Staubli VAL3: modIMM.pjx

--- modIMM.pjx ---
Parameters version=s7.2 stackSize=5000 millimeterUnit=true
Program file=_StartMachine.pgx
Program file=_WaitAuto.pgx
Program file=_WaitEnd.pgx
Program file=_WaitPart.pgx
Program file=_WaitPartDyn.pgx
Program file=BtRobotOff.pgx
Program file=checkMotStack.pgx
Program file=childAction.pgx
Program file=getSetting.pgx
Program file=IMMTiming.pgx
Program file=init.pgx
Program file=loadLibraries.pgx
Program file=primeAreaTest.pgx
Program file=primeMotStack.pgx
Program file=registerSetting.pgx
Program file=retrieveViews.pgx
Program file=runHigh.pgx
Program file=runLow.pgx
Program file=secuTask1.pgx
Program file=secuTask2.pgx
Program file=setDryRunSig.pgx
Program file=setSetting.pgx
Program file=slot.pgx
Program file=start.pgx
Program file=startAreaTest.pgx
Program file=stop.pgx
Program file=stopAreaTest.pgx
Program file=taskPartMade.pgx
Program file=updateView.pgx
Program file=WaitPart.pgx
Data file=modIMM.dtx
Library alias=io path=Disk://io/io.pjx
Library alias=SYS path=Disk://io_System/io_System.pjx
Library alias=scr path=Disk://Plastic/coreModules/modScreen/modScreen.pjx
Library alias=str path=Disk://Libraries/stringHandling/stringHandling.pjx
Library alias=lang path=Disk://Plastic/i18n/i18n.pjx
Library alias=debug path=Disk://Libraries/debug/debug.pjx
Library alias=data path=Disk://zData/zData.pjx
Library alias=status path=Disk://Plastic/coreModules/modStatusModel/modStatusModel.pjx
Library alias=EV path=Disk://Plastic/Consts/EVENT/EVENT.pjx
Library alias=sig path=Disk://Plastic/coreModules/modSignalSlot/modSignalSlot.pjx
Library alias=STATE path=Disk://Plastic/Consts/STATE/STATE.pjx
Library alias=views path=Disk://Plastic/coreModules/viewContainer/viewContainer.pjx
Library alias=jt path=Disk://Libraries/jointFunctions/jointFunctions.pjx
Type name=event path=Disk://Plastic/Types/event/event.pjx
Type name=settingType path=Disk://Plastic/Types/setting/setting.pjx
Type name=viewType path=Disk://Plastic/Types/view/view.pjx
Type name=childNodeType path=Disk://Plastic/Types/childNode/childNode.pjx
Type name=nodeType path=Disk://Plastic/Types/node/node.pjx

--- start.pgx ---
public program start()
begin
  // set nCaseBtRobOff to 1 instead of 0 in order to initialize the robot off function properly
  // If nCaseBtRobOff is 0 at start up it may happen that SYS:doRobotOff["+toString("",moduleIndex)+"] is on although btRobotOff assumes that
  // SYS:doRobotOff["+toString("",moduleIndex)+"] is off.

  call debug:setVerbosity(libPath(),debug:LEV_INFO)
  call loadLibraries()
  // call setDryRunSig(data:setDryRun)
  call sig:connect(EV:DRY_RUN,libPath())
  call sig:connect(EV:FATAL_ERROR,libPath())
  call sig:connect(EV:START_COMPLETE,libPath())
  call status:registerStatus(libPath(),status:CL_STATUS,"Wait for mould free condition","SYS:doMouldFree["+toString("",moduleIndex)+"]==true","SYS:doMouldFree["+toString("",moduleIndex)+"]==false",false,WAIT_MOULD_FREE,false)
  call status:registerStatus(libPath(),status:CL_STATUS,"Wait for mould open","SYS:diMouldOpen["+toString("",moduleIndex)+"]==true","SYS:diMouldOpen["+toString("",moduleIndex)+"]==false",false,WAIT_MOULD_OPEN,false)
  call status:registerStatus(libPath(),status:CL_STATUS,"Wait for robot enabled","SYS:doRobotOff["+toString("",moduleIndex)+"]==false","SYS:doRobotOff["+toString("",moduleIndex)+"]==true",false,WAIT_ROB_ENABLE,false)
  call status:registerStatus(libPath(),status:CL_STATUS,"Wait for IMM in auto mode","SYS:diMachineInAuto["+toString("",moduleIndex)+"]==true","SYS:diMachineInAuto["+toString("",moduleIndex)+"]==false",false,WAIT_ROB_ENABLE,false)
  call status:registerStatus(libPath(),status:CL_STATUS,"Wait for part produced","SYS:bPartMade["+toString("",moduleIndex)+"]==true","SYS:bPartMade["+toString("",moduleIndex)+"]==false",false,WAIT_PARTMADE,false)
  call status:registerStatus(libPath(),status:CL_ERROR,"Mould area test failed. Robot was not programmed to enter mould","","",true,AREA_TEST_FAIL,true)
  call status:registerStatus(libPath(),status:CL_ERROR,"Home position is defined in mould area","","",true,HOME_IN_MOULD,true)
  call status:registerStatus(libPath(),status:CL_ERROR,"Arm in mould while mould is not open","","",true,ARM_IN_MOULD_NO,true)
  call status:registerStatus(libPath(),status:CL_ERROR,"Arm in mould while 'Enable Closure' signal is set","","",true,ARM_IN_MOULD_ST,true)
end

--- _StartMachine.pgx ---
public program _StartMachine()
// Start machine cycle
  local bool bAreaTest
  local num nOldSpeedScale
  local bool bTestRun
  local string txt
  local num time
  local string sValue
begin
  //
  // add list of pending status messages
  //!i18n 16 -> "Wait for Mould Free Condition"

  call status:setEnabled(WAIT_MOULD_FREE,true)
  //!change 23.05.06, vdg: reduce speed in test mode when approaching the mould area boundary
  // from inside towards outside
  //!change 08.09.06, vdg: store data:setTestRun in a local variable
  bTestRun=data:setTestRun
  // prime the motion stack monitor which checks if the arm is actually
  // programmed to leave the mould when StartMachine() is called
  call primeMotStack()
  if bTestRun
    //wait(secu:nSafeZoneDist[0]<300)
    nOldSpeedScale=getMonitorSpeed()
    //!fix 09.06.06, vdg: set speed to the lower speed setting (current speedScale() or dry run speed)
    ///TODO
    //$setSpeed(min(speedScale(),10))
    //call setSpeed(min(getMonitorSpeed(),10))
    //wait(secu:nSafeZoneDist[0]<50)
    //$setSpeed(1)
    ///TODO
    //call setSpeed(1)
  endIf
  // WAIT GRIPPER OUT OF MOULD AREA ==================================================================================
  // record the safety distance of the robot

  time=clock()
  //requiredTime=0.2
  //currentTime=0
  // if (speedScale()>99) and (workingMode()==4) and (SYS:diMachineInAuto[moduleIndex]==true) and !bTestRun
  if (getMonitorSpeed()>99) and (workingMode()==4) and !bTestRun
    do
      // Check if there are still motions in the stack.
      // If it is empty, it means the robot never leaves the mould area before
      // StartMachine() is called.
      call checkMotStack()
    until (SYS:doMouldFree[moduleIndex]==true)
  else
    do
      // Check if there are still motions in the stack.
      // If it is empty, it means the robot never leaves the mould area before
      // StartMachine() is called.
      call checkMotStack()
    until (SYS:doMouldFree[moduleIndex]==true)
  endIf
  //
  call status:setEnabled(WAIT_MOULD_FREE,false)
  //
  //!change 18.05.06, vdg: check if doMouldFree has toggled
  call stopAreaTest(bAreaTest)
  // START MACHINE CYCLE =============================================================================================
  //!change 16.02.06, vdg: Allow to start IMM in endIf cycle mode SYS:bStartInEndCycl is set
  if (!SYS:CE_Requested or SYS:bStartInEndCycl) and !SYS:bPartMade[moduleIndex] and bAreaTest
    //!change 18.05.06, vdg: Stop robot at point where machine is being started
    //  and ask the user if it is safe to start the IMM
    if bTestRun
      bSuspendForTest=true
      // reset original speedScale only if speed was not modified by user meanwhile
      // wait for settled arm
      watch(isSettled(),3)
      // reset old speed setting if it wasn't changed by the user
      if getMonitorSpeed()==1
        ///TODO
        //$setSpeed(nOldSpeedScale)
        //call setSpeed(nOldSpeedScale)
      endIf
      //sValue=toString("4.0",secu:nSafeZoneDist[0])
      call str:printf((("Robot stopped approx. at point where IMM cycle is being started (Overshoot: %1mm). Press START to continue!")),sValue,txt)
      ///TODO
      //call ui:popUpCond(txt,"SYS:bBtStart==true",false)
      bSuspendForTest=true
      wait(bSuspendForTest==false)
    endIf
    //!change 08.06.06, vdg: Start IMM only if dry run mode is not active
    if !bTestRun
      SYS:doStartMachine[moduleIndex]=true
    endIf
    //call stat:stopTakeTime()
    //call stat:stopCycleTime()
    //call stat:startCycleTime()
    //call stat:startRobotTime()
  endIf
  //
end

--- _WaitAuto.pgx ---
public program _WaitAuto()
// Wait here until the machine is prepared to be started
begin
  // Enable Robot Off function........................................................
  bRobotOffAllow=true
  //
  //!change 18.06.05, vdg: Prime area test
  call primeAreaTest()
  //
  // ignore messages if in dry run mode
  if data:setDryRun==false
    call status:setEnabled(WAIT_IMM_AUTO,true)
  endIf
  call status:setEnabled(WAIT_MOULD_OPEN,true)
  call status:setEnabled(WAIT_ROB_ENABLE,true)
  // Stop the robot cycle time timer
  //call stat:stopRobotTime()
  // Wait machine in AUTO.............................................................
  do
    //Robot in position to be able use the Robot Off function.
    if SYS:diMachineInAuto[moduleIndex]==false and SYS:bRobotOffCalled[moduleIndex]
      bAtWaitPosition=true
    endIf
    //!change 08.06.06, vdg: ignore automatic signal in dry run mode
  until ((SYS:diMachineInAuto[moduleIndex]==true or data:setDryRun==true) and SYS:diMouldOpen[moduleIndex]==true and bRobotOff==false)
  //
  // Robot not in position to use Robot Off function..................................
  bAtWaitPosition=false
  //
  call status:setEnabled(WAIT_IMM_AUTO,false)
  call status:setEnabled(WAIT_MOULD_OPEN,false)
  call status:setEnabled(WAIT_ROB_ENABLE,false)
  //
  // Start measuring the take out time
  //call stat:startTakeTime()
  //
  call startAreaTest()
end

--- _WaitEnd.pgx ---
public program _WaitEnd()
// Halt robot here if "END" is activated
  local num nStateWaitEnd
begin
  // WAIT END OF CYCLE......................................................
  if SYS:CE_Requested and !SYS:bPartMade[moduleIndex] and SYS:doStartMachine[moduleIndex]==false
    do
      // Robot is running in production cycle (StateRobot==10)
      if SYS:nStateRobot==10 and isPowered() and SYS:diMachineInAuto[moduleIndex]==true
        // "End Of Cycle" running and no more parts in mould
        if SYS:CE_Requested and !SYS:bPartMade[moduleIndex] and SYS:diMachineInAuto[moduleIndex]==true
          nStateWaitEnd=30
        endIf
        // Robot Off called
        if SYS:bRobotOffCalled[moduleIndex]
          nStateWaitEnd=40
        endIf
      else
        // Robot or Machine not in AUTO
        if SYS:nStateRobot!=10
          nStateWaitEnd=0
        else
          // "End Of Cycle" running and no more parts in mould
          if SYS:CE_Requested and !SYS:bPartMade[moduleIndex] and SYS:CE_AtEndPos==false
            nStateWaitEnd=30
          endIf
          // Robot Off called
          if SYS:bRobotOffCalled[moduleIndex] and !bAtWaitPosition
            nStateWaitEnd=40
          endIf
        endIf
      endIf
      //
      switch (nStateWaitEnd)
        //
        //  Robot and Machine not in Auto.......................................
        case 0
          if SYS:diMachineInAuto[moduleIndex]==false
            //Wait Machine In Auto
            //user:sMessage[0]=user:sMessage[0]
          else
            //Wait [START] Robot
            //user:sMessage[0]=user:sMessage[0]
          endIf
        break
        //
        // "End Of Cycle" called and no more parts in mould.....................
        case 30
          if SYS:CE_Requested==true and SYS:bPartMade[moduleIndex]==false
            stopMove()
            wait(isSettled())
            SYS:CE_AtEndPos=true
            delay(0)
          endIf
        break
        //
        // Robot Off called.......................................................
        case 40
          wait(isSettled())
          stopMove()
          bAtWaitPosition=true
          delay(0)
        break
      endSwitch
      //
      // Wait until robot is at end position......................................
    until (SYS:CE_AtEndPos==true or bAtWaitPosition==true and isSettled())
    //
    // Reset StartMachine.................................................................................................
    SYS:doStartMachine[moduleIndex]=false
  endIf
end

--- _WaitPartDyn.pgx ---
public program _WaitPartDyn()
// Wait part made in machine and mould fully open
begin
  //!brief
  // Wait for a part being made and conditions for the robot to enter mold.
  //
  call WaitPart(true)
end

--- init.pgx ---
public program init()
  local bool ok
  local string path
  local num idx
begin
  // set module index
  path=libPath()
  path=right(path,1)
  path=toNum(path,moduleIndex,ok)
  if !ok
    moduleIndex=0
  endIf
  name="IMM"+toString("1.0",moduleIndex)
  IMM_IO_PTH="2:IO/1:"+name
  nCaseBtRobOff=1
  bState=false
  pointer=0
  for idx=0 to size(timings)-1
    timings[idx]=0
  endFor

end

--- loadLibraries.pgx ---
program loadLibraries()
begin
//  nResult=scr:libLoad("Plastic/Modules/modScreen.zip","a81d706f651db0a6b2")
//  if nResult!=0
//    name=libPath()
//    nResult=scr:libLoad("Plastic/Modules/modScreen")
//    if nResult!=0
//      popUpMsg(name+":  Problem loading library for scr:")
//      call debug:error(libPath(),": Problem loading library for scr:")
//    else
//      call debug:info(libPath(),": Loading uncrypted version "+scr:libPath())
//    endIf
//  endIf
  // SECU
//  nResult=secu:libLoad("Plastic/Modules/modSafety.zip","a81d706f651db0a6b2")
//  if nResult!=0
//    name=libPath()
//    nResult=secu:libLoad("Plastic/Modules/modSafety")
//    if nResult!=0
//      popUpMsg(name+":  Problem loading library for secu:")
//      call debug:error(libPath(),": Problem loading library for secu:")
//    else
//      call debug:info(libPath(),": Loading uncrypted version "+secu:libPath())
//    endIf
//  endIf
//  // STATUS
//  nResult=stat:libLoad("Plastic/Modules/modStatus.zip","a81d706f651db0a6b2")
//  if nResult!=0
//    name=libPath()
//    nResult=stat:libLoad("Plastic/Modules/modStatus")
//    if nResult!=0
//      popUpMsg(name+":  Problem loading library for stat:")
//      call debug:error(libPath(),": Problem loading library for stat:")
//    else
//      call debug:info(libPath(),": Loading uncrypted version "+stat:libPath())
//    endIf
//  endIf
end

--- primeAreaTest.pgx ---
public program primeAreaTest()
begin
  // reset test state machine
  nAreaTestState=0
end

--- retrieveViews.pgx ---
public program retrieveViews(viewType& view_, num& idx_)
begin
  switch idx_
    case 0
      view_.path=IMM_IO_PTH
      view_.label="IMM"
      call views:appendNode(view_.nodes,"Safety")
      call views:appendNode(view_.nodes,"Machine")
      call views:appendNode(view_.nodes,"Ejectors")
      call views:appendNode(view_.nodes,"Cores")
      call views:appendNode(view_.nodes,"Mould")
      view_.type=view_.TYPE_TREEVIEW
    break
  endSwitch
end

--- run.pgx ---
public program run()
begin
  call taskPartMade()
  call IMMTiming()
end

--- runHigh.pgx ---
public program runHigh()
begin
  call taskPartMade()
  call IMMTiming()
   call BtRobotOff()

  call secuTask1()
  call secuTask2()
end

--- secuTask1.pgx ---
public program secuTask1()
// Control "Mould Area Free" from robot
  local point pLocFlange
  local point pLocTCP
begin
  //
  //!change 23.04.06, vdg: added global variable that contains the distance to the safety zone
  // Security zon in millimeter for wrist relativ to IMM Backside...........
  // nSafeZon[0]=300
  //
  // LOOP: task "RobSafe1"..................................................

    //
    // Get current robot position relative to the frame of IMM Backside.....
    pLocFlange=here(flange,data:fAreaIMM)
    pLocTCP=here(data:tTCP,data:fAreaIMM)
    //
    // Set signal "Mould Area Free" to machine..............................
    nMouldAreaDist=max(pLocTCP.trsf.z,pLocFlange.trsf.z)-nMouldAreaZone
    SYS:doMouldFree[moduleIndex]=nMouldAreaDist<0
    //
    if SYS:doMouldFree==false
      SYS:doStartMachine=false
      bRobotOff=false
    endIf
    //
    //!change 18.05.06, vdg: Test if MouldFree Signal has toggled while robot was in mould
    switch nAreaTestState
      // initialize test
      case 0
        //nAreaTestState=0
        //bAreaFlag=SYS:doMouldFree
      break
      // wait for high state
      case 10
        if SYS:doMouldFree==true
          nAreaTestState=20
        endIf
      break
      // wait for low state
      case 20
        if SYS:doMouldFree==false
          nAreaTestState=30
        endIf
      break
      // wait for high state again
      case 30
        if SYS:doMouldFree==true
          nAreaTestState=40
        endIf
      break
      // final state
      // this state must be reached when startIMM() is called
      case 40
      break
    endSwitch
//  SYS:doSecu[0]=false
//  SYS:doSecu[1]=false
end

--- secuTask2.pgx ---
public program secuTask2()
// Control of Safety realay
  local point pLocFlange
  local point pLocTCP
begin
  // wait until system is initialized
  if SYS:nStateRobot<=STATE:INITIALIZING
    return
  endIf
  if SYS:doSecu[0]==false or SYS:doSecu[1]==false
    return
  endIf
  // Get home position relative to the frame of IMM mould area.....
  if jt:isTXRobot
    pLocFlange=jointToPoint(flange,data:fAreaIMM,data:jHomeTX)
    pLocTCP=jointToPoint(data:tTCP,data:fAreaIMM,data:jHomeTX)
  else
    pLocFlange=jointToPoint(flange,data:fAreaIMM,data:jHomeTS)
    pLocTCP=jointToPoint(data:tTCP,data:fAreaIMM,data:jHomeTS)
  endIf
//
  if pLocTCP.trsf.z>nMouldAreaZone
    call status:raise(HOME_IN_MOULD,"")
  endIf
  // Get current robot position relative to the frame of IMM Backside.....
  pLocFlange=here(flange,data:fAreaIMM)
  pLocTCP=here(data:tTCP,data:fAreaIMM)
  nMouldAreaDist=max(pLocTCP.trsf.z,pLocFlange.trsf.z)-nMouldAreaZone
  //
  // Robotarm in mould when sig:MouldOpen missing or sig:StartIMM is active..........................................................
  if SYS:doMouldFree==false and (SYS:diMouldMidOpen==false and SYS:diMouldOpen==false)
    call status:raise(ARM_IN_MOULD_NO,"")
  endIf
  if (SYS:doMouldFree==false and SYS:doStartMachine==true)
    call status:raise(ARM_IN_MOULD_ST,"")
  endIf
end

--- setDryRunSig.pgx ---
public program setDryRunSig(bool enable_)
begin
  if enable_
    call debug:warning(libPath(),"Dry run mode enabled")
    dioLink(SYS:diEjcIn,SYS:doEjcIn)
    dioLink(SYS:diEjcOut,SYS:doEjcOut)
    dioLink(SYS:diCore1Pos1,SYS:doCore1Pos1)
    dioLink(SYS:diCore1Pos2,SYS:doCore1Pos2)
    dioLink(SYS:diCore2Pos1,SYS:doCore2Pos1)
    dioLink(SYS:diCore2Pos2,SYS:doCore2Pos2)
  else
    call debug:warning(libPath(),"Dry run mode disabled")
    call SYS:InitSysIO()
  endIf
end

--- slot.pgx ---
public program slot(event& event_)
begin
  switch event_.nType
    case EV:DRY_RUN
      call setDryRunSig(event_.sParam=="1")
    break
    case EV:START_COMPLETE
      SYS:doSecu[0]=true
    SYS:doSecu[1]=true
    break
  endSwitch
end

--- stopAreaTest.pgx ---
public program stopAreaTest(bool& bResult_[])
begin
  // test result of area test state machine
  // the state nAreaTestState must be 40
  if nAreaTestState!=40 and nAreaTestState!=0
    call status:raise(AREA_TEST_FAIL,"")
  endIf
  bResult_=nAreaTestState==40 or nAreaTestState==0
end

--- taskPartMade.pgx ---
program taskPartMade()
// Part produced in an IMM
begin
  // Conditions for part made is registered in program.
  // Arm will enter mould. Close mould is not allowed.
  if !bRobotOffAllow
    SYS:doStartMachine[moduleIndex]=false
  endIf
  if SYS:doMouldFree[moduleIndex]==false or SYS:bRobotHome
    bRobotOffAllow=true
  endIf
  // RESET StartMachine.......................................................
  // handle reset according to given IMM type
  switch nImmType
    // standard IMM, e.g. Netstal
    case 0
      // reset doStartMachine when IMM is switched to manual
      if SYS:diMachineInAuto[moduleIndex]==false
        SYS:doStartMachine[moduleIndex]=false
      endIf
      // set robot off signal to IMM
      SYS:doRobotOff[moduleIndex]=bRobotOff
    break
    // IMMs of type 1, that need special treatment of doStartIMM, e.g. Negri Bossi
    case 1
      // reset doStartMachine when IMM is switched to manual and handling is disabled
      if SYS:diMachineInAuto[moduleIndex]==false and SYS:doRobotOff[moduleIndex]==false
        SYS:doStartMachine[moduleIndex]=false
      endIf
      if bRobotOff==true
        // Disable doStartMachine and doRobotOff if the robot is approaching the mold
        // The distance 20mm is set in order to have a pre warning before the arm
        // actually enters the mold area.
        if nMouldAreaDist>-20
          SYS:doStartMachine[moduleIndex]=false
          SYS:doRobotOff[moduleIndex]=false
        else
          SYS:doStartMachine[moduleIndex]=true
          // set robot off signal to IMM
          SYS:doRobotOff[moduleIndex]=bRobotOff
        endIf
      else
        // set robot off signal to IMM
        SYS:doRobotOff[moduleIndex]=bRobotOff
      endIf
    break
  endSwitch

  // RESET PartMade (Ejecor and "Robot OFF")..................................
  if SYS:diMachineInAuto[moduleIndex]==false or bRobotOff==true
    if SYS:diMachineInAuto[moduleIndex]==false
      SYS:doEjcIn=true
      SYS:doEjcOut=true
    else
      SYS:doEjcIn=false
      SYS:doEjcOut=false
    endIf
    switch nStateRstPart[0]
      case 0
        if (SYS:diEjcOut==true and SYS:diEjcIn==false)
          nStateRstPart[0]=1
        endIf
      break
      case 1
        if (SYS:diEjcOut==false and SYS:diEjcIn==true)
          SYS:bPartMade[moduleIndex]=false
          nStateRstPart[0]=0
        endIf
      break
    endSwitch
  else
    nStateRstPart[0]=0
  endIf
  //
  // RESET PartMade (Core and "Robot OFF")...................................
  if SYS:diMachineInAuto[moduleIndex]==false or bRobotOff==true
    if SYS:diMachineInAuto[moduleIndex]==false
      SYS:doCore1Pos1=true
      SYS:doCore1Pos2=true
    else
      SYS:doCore1Pos1=false
      SYS:doCore1Pos2=false
    endIf
    switch nStateRstPart[1]
      case 0
        if (SYS:diCore1Pos2==true and SYS:diCore1Pos1==false)
          nStateRstPart[1]=1
        endIf
      break
      case 1
        if (SYS:diCore1Pos2==false and SYS:diCore1Pos1==true)
          SYS:bPartMade[moduleIndex]=false
          nStateRstPart[1]=0
        endIf
      break
    endSwitch
  else
    nStateRstPart[1]=0
  endIf
  //
  // RESET PartMade (machine goes from manual mode to auto)..................
  switch nStateRstPart[3]
    case 0
      if (SYS:diMachineInAuto[moduleIndex]==false)
        nStateRstPart[3]=1
      endIf
    break
    case 1
      if (SYS:diMachineInAuto[moduleIndex]==true)
        SYS:bPartMade[moduleIndex]=false
        SYS:doEjcIn=false
        SYS:doEjcOut=false
        SYS:doCore1Pos1=false
        SYS:doCore1Pos2=false
        nStateRstPart[3]=0
      endIf
    break
  endSwitch
  //
  // PART MADE.............................................................
  switch nStatePartMade
    // Mould open
    case 0
      if (SYS:bPartMade[moduleIndex]==false and SYS:diMouldOpen[moduleIndex]==true and SYS:diMachineInAuto[moduleIndex]==true)
        nStatePartMade=1
        // count parts
        data:cyclesProduced=data:cyclesProduced+1
        if SYS:diRejectPart==true
          data:cyclesRejected=data:cyclesRejected+1
        endIf
      endIf
    break
    // Mould is closing
    case 1
      if SYS:diMouldOpen[moduleIndex]==false and SYS:diMachineInAuto[moduleIndex]==true
        nStatePartMade=2
      endIf
    break
    // Mould closed
    case 2
      if SYS:diMouldClosed[moduleIndex]==true and SYS:diMachineInAuto[moduleIndex]==true
        SYS:bPartMade[moduleIndex]=true
        // Reset of ejector signals disabled here, as some IMMs
        // have problems when ejector signal is reset when mould is closed as the ejectors
        // are not held in position actively anymore (due to leacking valve or similar).
        // Instead the ejector signals are reset when the mould starts opening again
        // (see state 3)
        //SYS:doEjcIn=false
        //SYS:doEjcOut=false
        SYS:doStartMachine[moduleIndex]=false
        nStatePartMade=3
      endIf
      // Mould was never closed
      if SYS:diMouldOpen[moduleIndex]==true and SYS:diMachineInAuto[moduleIndex]==true
        nStatePartMade=0
      endIf
    break
    // Mould starts opening
    case 3
      if SYS:diMouldClosed[moduleIndex]==false and SYS:diMachineInAuto[moduleIndex]==true
        SYS:doEjcIn=false
        SYS:doEjcOut=false
        nStatePartMade=0
      endIf
      // Mould was never closed
      if SYS:diMouldOpen[moduleIndex]==true and SYS:diMachineInAuto[moduleIndex]==true
        nStatePartMade=0
      endIf
    break
  endSwitch
end

--- updateView.pgx ---
public program updateView()
  local string sValues[5]
  local childNodeType child
begin

  call views:childDIO(views:views[IMM_IO_PTH].nodes[0],0,"Safety Relay 1",SYS:doSecu[0])
  call views:childDIO(views:views[IMM_IO_PTH].nodes[0],1,"Safety Relay 2",SYS:doSecu[1])

  sValues[0]=toString("4.0",nMouldAreaDist)
  if SYS:doMouldFree[moduleIndex]==true
    sValues[1]="/ti"
  endIf
  call str:printf(("%2 %1/tnmm"),sValues,child.valueText)
  child.label="Safety Distance"
  call views:setChild(views:views[IMM_IO_PTH].nodes[0],2,child)

  call views:childDIO(views:views[IMM_IO_PTH].nodes[1],0,"Robot Off",SYS:doRobotOff[moduleIndex])
  call views:childDIO(views:views[IMM_IO_PTH].nodes[1],1,"Mould Area Free",SYS:doMouldFree[moduleIndex])
  call views:childDIO(views:views[IMM_IO_PTH].nodes[1],2,"Enable Mould Closure",SYS:doStartMachine[moduleIndex])
  call views:childDIO(views:views[IMM_IO_PTH].nodes[1],3,"Automatic Mode",SYS:diMachineInAuto[moduleIndex])
  call views:childDIO(views:views[IMM_IO_PTH].nodes[1],4,"Reject Part",SYS:diRejectPart[moduleIndex])

  call views:childDIO(views:views[IMM_IO_PTH].nodes[2],0,"Ejector forward",SYS:doEjcOut[moduleIndex])
  call views:childDIO(views:views[IMM_IO_PTH].nodes[2],1," ",SYS:diEjcOut[moduleIndex])
  call views:childDIO(views:views[IMM_IO_PTH].nodes[2],2,"Ejector forward",SYS:doEjcIn[moduleIndex])
  call views:childDIO(views:views[IMM_IO_PTH].nodes[2],3," ",SYS:diEjcIn[moduleIndex])

  call views:childDIO(views:views[IMM_IO_PTH].nodes[3],0,"Core 1 Pos 1",SYS:doCore1Pos1[moduleIndex])
  call views:childDIO(views:views[IMM_IO_PTH].nodes[3],1," ",SYS:diCore1Pos1[moduleIndex])
  call views:childDIO(views:views[IMM_IO_PTH].nodes[3],2,"Core 1 Pos 2",SYS:doCore1Pos2[moduleIndex])
  call views:childDIO(views:views[IMM_IO_PTH].nodes[3],3," ",SYS:diCore1Pos2[moduleIndex])
  call views:childDIO(views:views[IMM_IO_PTH].nodes[3],4,"Core 2 Pos 1",SYS:doCore2Pos1[moduleIndex])
  call views:childDIO(views:views[IMM_IO_PTH].nodes[3],5," ",SYS:diCore1Pos1[moduleIndex])
  call views:childDIO(views:views[IMM_IO_PTH].nodes[3],6,"Core 2 Pos 2",SYS:doCore2Pos2[moduleIndex])
  call views:childDIO(views:views[IMM_IO_PTH].nodes[3],7," ",SYS:diCore1Pos2[moduleIndex])


  call views:childDIO(views:views[IMM_IO_PTH].nodes[4],0,"Mould Open",SYS:doFullOpening[moduleIndex])
  call views:childDIO(views:views[IMM_IO_PTH].nodes[4],1," ",SYS:diMouldOpen[moduleIndex])
  call views:childDIO(views:views[IMM_IO_PTH].nodes[4],2,"Mould Closed",SYS:diMouldClosed[moduleIndex])
  call views:childDIO(views:views[IMM_IO_PTH].nodes[4],3,"Mould Intermediate Pos",SYS:diMouldMidOpen[moduleIndex])
end

--- WaitPart.pgx ---
program WaitPart(bool bMode_)
// Wait part made in machine and mould fully open
  local num nStateWaitPart
  local num nCaseManAuto
  local bool bFirstRun
  local bool exitCondition
begin
  //!brief
  // Wait for a part being made and conditions for the robot to enter mold.
  //
  //!param bMode : If bMode is true, dynamic mode is used
  //
  //!change 07.04.06, vdg: added parameter bMode_ for dynamic wait part function.
  //                       WaitPartDynamic() is therefore obsolete.
  // WAIT PART....................................................................................
  //!change 18.06.05, vdg: Prime area test
  //call secu:primeAreaTest()
  //
  bRobotOffAllow=true
  bFirstRun=true
  //
  call status:setEnabled(WAIT_MOULD_OPEN,true)
  call status:setEnabled(WAIT_ROB_ENABLE,true)
  // ignore messages if in dry run mode
  if data:setDryRun==false
    call status:setEnabled(WAIT_IMM_AUTO,true)
    call status:setEnabled(WAIT_PARTMADE,true)
  endIf
  //
  //!change 07.07.07, vdg: stop the robot cycle time timer
  //call stat:stopRobotTime()
  do
    // Robot is running in production cycle (StateRobot==10)
    if SYS:nStateRobot==10 and SYS:diMachineInAuto[moduleIndex]==true
      nCaseManAuto=0
      // Wait part produced
      if !SYS:bPartMade[moduleIndex] or SYS:diMouldOpen[moduleIndex]==false
        nStateWaitPart=10
      endIf
      // No part is produced, Start Machine
      if !SYS:bPartMade[moduleIndex] and !SYS:CE_Requested and SYS:diMouldOpen[moduleIndex]==true and SYS:diMachineInAuto[moduleIndex]==true
        nStateWaitPart=20
      endIf
      // "End Of Cycle" running and no more parts in mould
      if SYS:CE_Requested and !SYS:bPartMade[moduleIndex] and SYS:diMachineInAuto[moduleIndex]==true
        nStateWaitPart=30
      endIf
      // Robot Off called
      if SYS:bRobotOffCalled[moduleIndex]
        nStateWaitPart=40
      endIf
    else
      // Machine not in AUTO...........................................
      if SYS:nStateRobot!=10
        nStateWaitPart=0
      else
        if SYS:CE_Requested or SYS:bRobotOffCalled[moduleIndex]
          // "End Of Cycle" running and no more parts in mould
          if SYS:CE_Requested and !SYS:bPartMade[moduleIndex] and SYS:CE_AtEndPos==false
            nStateWaitPart=30
          endIf
          // Robot Off called
          if SYS:bRobotOffCalled[moduleIndex] and !bAtWaitPosition
            nStateWaitPart=40
          endIf
        else
          nStateWaitPart=0
        endIf
      endIf
    endIf
    //
    switch (nStateWaitPart)
      //
      // Machine not in Auto...................................................
      case 0
        if SYS:diMachineInAuto[moduleIndex]==false
          //Wait Machine In Auto
          //user:sMessage[0]=user:sMessage[0]
        else
          //Wait [START] Robot
          //user:sMessage[0]=user:sMessage[0]
        endIf
        switch nCaseManAuto
          // Wait machine in manual mode
          case 0
            if SYS:diMachineInAuto[moduleIndex]==false
              nCaseManAuto=1
            endIf
          break
          // Wait machine in Auto
          case 1
            if SYS:diMachineInAuto[moduleIndex]==true and !SYS:bPartMade[moduleIndex]
              // Start machine cycle
              //!change 08.06.06, vdg: do not start IMM in dry run mode
              if (SYS:doMouldFree[moduleIndex]==true) and !data:setDryRun
                SYS:doStartMachine[moduleIndex]=true
              endIf
              nCaseManAuto=0
            endIf
          break
        endSwitch
      break
      //
      // Wait part produced
      case 10
        //Wait PART
        //user:sMessage[0]=user:sMessage[0]
      break
      //
      // Start Machine if no part is made..............................................................................
      case 20
        // Start Machine
        //user:sMessage[0]=user:sMessage[0]
        // Gripper out of mould area
        if (SYS:doMouldFree[moduleIndex]==true)
          // Start machine cycle
          if SYS:CE_Requested==false and SYS:diMachineInAuto[moduleIndex]==true
            //!change 18.05.06, vdg: Stop robot at point where machine is being started
            //  and ask the user if it is safe to start the IMM
            //
            // only stop the robot if test run is activated and this is the first
            // cycle of WaitPart()
            if data:setTestRun and bFirstRun
              bFirstRun=false
              // wait until no motion is pending in the motion stack
              // the arm should then be at the waiting position in front of the mould
              wait(isEmpty())
              //!todo: make displayed message nicer
              //!i18n 23 -> "Robot stopped approx. at point where IMM cycle is being started. Press START to continue!"
              ///TODO
              //call ui:popUpCond((("Robot stopped approx. at point where IMM cycle is being started. Press START to continue!")),"SYS:bBtStart==true",false)
              // send request to robMotionCtrl to stop the arm
              bSuspendForTest=true
              wait(bSuspendForTest==false)
            endIf
            //!change 08.06.06, vdg: do not start IMM in dry run mode
            if !data:setDryRun
              SYS:doStartMachine[moduleIndex]=true
            endIf
          endIf
        endIf
      break
      //
      // "End Of Cycle" called and no more parts in mould.............................................................
      case 30
        if SYS:CE_Requested==true and SYS:bPartMade[moduleIndex]==false
          SYS:CE_AtEndPos=true
          delay(0)
        endIf
      break
      //
      // Robot Off called.................................................................................................................................................
      case 40
        bAtWaitPosition=true
        delay(0)
      break
    endSwitch
    //
    // Wait until part is made and conditon to enter mould is true........................................................................................................
    //!change 08.06.06, vdg: ignore autmatic signal and part made flag in dry run mode
    exitCondition=(SYS:bPartMade[moduleIndex] or data:setDryRun) and ((SYS:diMouldMidOpen[moduleIndex]==true and bMode_) or SYS:diMouldOpen[moduleIndex]==true)
    exitCondition=exitCondition and (SYS:diMachineInAuto[moduleIndex]==true or data:setDryRun) and bRobotOff==false and SYS:nStateRobot==10 and isPowered()
  until exitCondition
  //
  //
  // Reset StartMachine.................................................................................................
  SYS:doStartMachine[moduleIndex]=false
  //
  // Robot is allowed to go inside mould area. Do not close mould until arm has entered mould area.
  bRobotOffAllow=false
  //
  // Start measuring the take out time
  //call stat:startTakeTime()
  //
  //!change 18.06.05, vdg: Start area test
  call startAreaTest()
  call status:setEnabled(WAIT_IMM_AUTO,false)
  call status:setEnabled(WAIT_MOULD_OPEN,false)
  call status:setEnabled(WAIT_ROB_ENABLE,false)
  call status:setEnabled(WAIT_PARTMADE,false)
  // reset move ID counter only at first IMM
  if moduleIndex==0
    setMoveId(0)
  endIf
end
